(* IEC 61131-3 sources: programs/VI-54/VI-54_20171205/VI-54_20171205/Stations/PLC_VI54/VI-54_171014/Class/CurrentWatcher, 1 file *)

(* ---- CurrentWatcher.st ---- *)
(*!
<Class
	Name               = "CurrentWatcher"
	Revision           = "0.0"
	RealtimeTask       = "false"
	CyclicTask         = "true"
	BackgroundTask     = "false"
	Sigmatek           = "false"
	OSInterface        = "false"
	HighPriority       = "false"
	Automatic          = "false"
	UpdateMode         = "Prescan"
	SharedCommandTable = "true"
	Objectsize         = "(600,480)">
	<Channels>
		<Server Name="ActCurrent" Visualized="true" Initialize="false" WriteProtected="true" Retentive="false"/>
		<Server Name="CheckCurrent" Visualized="true" Initialize="true" WriteProtected="false" Retentive="File"/>
		<Server Name="ClassSvr" Visualized="true" Remotely="true" Initialize="false" WriteProtected="false" Retentive="false"/>
		<Server Name="MaxCurrent" Visualized="true" Initialize="false" WriteProtected="true" Retentive="false"/>
		<Server Name="ResetErrors" Visualized="true" Initialize="false" WriteProtected="false" Retentive="false"/>
		<Server Name="StallCurrent" Visualized="true" Initialize="false" WriteProtected="true" Retentive="false"/>
		<Server Name="TypeOfCheck" Visualized="true" Initialize="true" WriteProtected="false" Retentive="File"/>
		<Client Name="_DriveASyncPara1" Required="true" Internal="true"/>
		<Client Name="CurrentToHigh" Required="true" Internal="true"/>
		<Client Name="DriveAxis" Required="true" Internal="false" Comment="object channel to the class _DriveAxis"/>
		<Client Name="LmcAxic" Required="true" Internal="false"/>
	</Channels>
	<Network Name="CurrentWatcher">
		<!-- List of Components in this network -->
		<Components>
			<Object
				Name       = "_DriveASyncPara1"
				Class      = "_DriveASyncPara"
				Position   = "(270,180)"
				Visualized = "true">
				<Channels>
					<Server Name="ErrorQuit"/>
					<Server Name="ParaNr"/>
					<Server Name="ParaRdWr"/>
					<Server Name="ParaValue"/>
					<Server Name="State"/>
					<Client Name="DriveAxis"/>
					<Client Name="ErrorCode"/>
				</Channels>
			</Object>
			<Object
				Name       = "CurrentToHigh"
				Class      = "_AlarmX0Para"
				Position   = "(270,570)"
				Visualized = "true">
				<Channels>
					<Server Name="ClassSvr"/>
					<Client Name="Acknow"/>
					<Client Name="Config" Value="0"/>
					<Client Name="Group"/>
				</Channels>
			</Object>
		</Components>
		<Comments>
		</Comments>
		<!-- List of Connections in this network -->
		<Connections>
			<Connection Source="this._DriveASyncPara1" Destination="_DriveASyncPara1.State"/>
			<Connection Source="_DriveASyncPara1.DriveAxis" Destination="this.DriveAxis" Vertices="(270,270),(38,270),"/>
			<Connection Source="this.CurrentToHigh" Destination="CurrentToHigh.ClassSvr"/>
			<Connection Source="this.ClassSvr" Destination="CurrentToHigh.ClassSvr" Vertices="(788,570),(570,660),"/>
		</Connections>
		<!-- Headerfiles -->
		<Options>
		</Options>
	</Network>
</Class>
*)
CurrentWatcher : CLASS
	TYPE
#pragma pack(push, 1)
	  CurrentTypes : STRUCT
	    StallCurrent : DINT;
	    MaxCurrent : DINT;
	    ActCurrent : DINT;
	  END_STRUCT;
#pragma pack(pop)
	END_TYPE
  //Servers:
	CheckCurrent 	: SvrChCmd_DINT;
	TypeOfCheck 	: SvrCh_SoortCheck;
	StallCurrent 	: SvrCh_DINT;
	MaxCurrent 	: SvrCh_DINT;
	ActCurrent 	: SvrCh_DINT;
	ResetErrors 	: SvrCh_DINT;
	ClassSvr 	: SvrCh_DINT;
  //Clients:
	LmcAxic 	: CltChCmd__LMCAxis;
	DriveAxis 	: CltChCmd__DriveAxisBase;
	_DriveASyncPara1 	: CltChCmd__DriveASyncPara;
	CurrentToHigh 	: CltChCmd__AlarmX0Para;
  //Variables:
		CurrentValues 	: CurrentTypes;
		CurrentToHighTmr 	: UDINT;
		TmrOlineAlignment 	: UDINT;
		ReadCurrent 	: DINT;
		LmcAxisState 	: _LMCAXIS_STATUS;
		ResetEenmaal 	: DINT;
  //Functions:

	FUNCTION VIRTUAL GLOBAL CyWork
		VAR_INPUT
			EAX 	: UDINT;
		END_VAR
		VAR_OUTPUT
			state (EAX) 	: UDINT;
		END_VAR;

	FUNCTION GLOBAL ResetError;

	FUNCTION GLOBAL ReadCurrents;

	FUNCTION VIRTUAL GLOBAL ClassSvr::Read
		VAR_OUTPUT
			output (EAX) 	: DINT;
		END_VAR;

	FUNCTION VIRTUAL GLOBAL ClassSvr::Write
		VAR_INPUT
			input (EAX) 	: DINT;
		END_VAR
		VAR_OUTPUT
			result (EAX) 	: DINT;
		END_VAR;
  //Tables:
	FUNCTION @STD
		VAR_OUTPUT
			ret_code	: CONFSTATES;
		END_VAR;
	FUNCTION GLOBAL TAB @CT_;
END_CLASS;

#pragma using _AlarmX0Para
#pragma using _DriveASyncPara
#pragma usingLtd _DriveAxisBase
#pragma usingLtd _LMCAxis

FUNCTION VIRTUAL GLOBAL CurrentWatcher::CyWork
	VAR_INPUT
		EAX 	: UDINT;
	END_VAR
	VAR_OUTPUT
		state (EAX) 	: UDINT;
	END_VAR

  // controleerd of de homesensor niet kapot is
  // Dus de stroom mag niet te hoog oplopen!

  // Lees statussen uit
  ReadCurrents();
  LmcAxic       := LmcAxic.Read();
  LmcAxisState  := LmcAxic.ReadAxisStatus();
  MaxCurrent    := CurrentValues.MaxCurrent;
  StallCurrent  := CurrentValues.StallCurrent;
  ActCurrent    := CurrentValues.ActCurrent;

  // kijk of ingevulde stroom groter is dan '100' mA, anders neem max stroom / 4
  if CheckCurrent <= 100 & CurrentValues.MaxCurrent > 0 then
    CheckCurrent := (CurrentValues.MaxCurrent / 4); // rond de 1 Amp gezekerd wanneer er niks wordt ingevuld
  end_if;

  // Verschillende types die gechecked kunnen worden
  if TypeOfCheck = HomeCheck then
    if LmcAxisState.IsReferenced = 0 then // Alleen checken bij homen
      if CurrentValues.ActCurrent > CheckCurrent then
        if (ops.tAbsolute - CurrentToHighTmr) >= 5 * _10ms then
          LmcAxic.PowerOff(Mode:=LMCAXIS_IMMEDIATE_STOPP);
          CurrentToHigh.ClassSvr.Write(input:= 1);
        end_if;
      else
        CurrentToHighTmr := ops.tAbsolute;
      end_if;
    end_if;
  elsif TypeOfCheck = MoveCheck then
    if LmcAxic = MOVE_LMCAXIS then // Alleen checken bij moving
      if CurrentValues.ActCurrent > CheckCurrent then
        if (ops.tAbsolute - CurrentToHighTmr) >= 5 * _10ms then
          LmcAxic.PowerOff(Mode:=LMCAXIS_IMMEDIATE_STOPP);
          CurrentToHigh.ClassSvr.Write(input:= 1);
        end_if;
      else
        CurrentToHighTmr := ops.tAbsolute;
      end_if;
    end_if;
  end_if;

  // Resetten
  if ResetErrors = 1 then
    if ResetEenmaal = 0 then
      ResetError();
      ResetEenmaal := 1;
    end_if;
  else
    ResetEenmaal := 0;
  end_if;

	state := READY;

END_FUNCTION

FUNCTION GLOBAL CurrentWatcher::ResetError

  // Reset home error
  CurrentToHigh.ClassSvr.Write(input:= 0);

END_FUNCTION

FUNCTION GLOBAL CurrentWatcher::ReadCurrents

  // Lees stromen uit
  if DriveAxis.IsOnline() = 1 then
    if ops.tAbsolute - TmrOlineAlignment >= 1000 then
      if CurrentValues.StallCurrent = 0 then
        _DriveASyncPara1.ParaRdWr.Write(0);
        _DriveASyncPara1.ParaNr.Write(56);  // Stall current of the motor (rms).
        if ops.tAbsolute - TmrOlineAlignment >= 1100 then
          CurrentValues.StallCurrent := _DriveASyncPara1.ParaValue.Read();
          TmrOlineAlignment := ops.tAbsolute;
        end_if;
      elsif CurrentValues.MaxCurrent = 0 then
        _DriveASyncPara1.ParaRdWr.Write(0);
        _DriveASyncPara1.ParaNr.Write(57);  // Maximum current of the motor (rms).
        if ops.tAbsolute - TmrOlineAlignment >= 1100 then
          CurrentValues.MaxCurrent := _DriveASyncPara1.ParaValue.Read();
          TmrOlineAlignment := ops.tAbsolute;
        end_if;
      else
        _DriveASyncPara1.ParaRdWr.Write(0);
        _DriveASyncPara1.ParaNr.Write(191);  // Actual current of the motor.
        CurrentValues.ActCurrent := ABS(_DriveASyncPara1.ParaValue.Read());
      end_if;
    end_if;
  end_if;

END_FUNCTION

FUNCTION VIRTUAL GLOBAL CurrentWatcher::ClassSvr::Read
	VAR_OUTPUT
		output (EAX) 	: DINT;
	END_VAR

	ClassSvr := CurrentToHigh.ClassSvr.Read();
	output := ClassSvr;

END_FUNCTION

FUNCTION VIRTUAL GLOBAL CurrentWatcher::ClassSvr::Write
	VAR_INPUT
		input (EAX) 	: DINT;
	END_VAR
	VAR_OUTPUT
		result (EAX) 	: DINT;
	END_VAR

	ClassSvr := input;
	result := (CurrentToHigh.ClassSvr.Write(ClassSvr))$DINT;

END_FUNCTION
